SUBAPPLICATION Uebung_011f_ROUND_AR_AX (* Wie Uebung_011f_AX, aber mit OSCAT ROUND_AR dazwischen (rundet auf N Nachkommastellen) *)
  (* Standard: 61499-2; Description: Copyright (c) 2026 Meisterschulen am Ostbahnhof This program and the accompanying materials are made available under the terms of the Eclipse Public License 2.0 which is available at https://www.eclipse.org/legal/epl-2.0/ SPDX-License-Identifier: EPL-2.0 *)
  (* Version 1.0, 2026-10-09, Franz Höpfinger, Meisterschulen am Ostbahnhof, initial API and implementation and/or initial documentation *)
  PACKAGE Uebungen;
  IMPORT Uebungen::const::UT::DefaultPool_Numeric::InputNumber_I3_N;
  IMPORT Uebungen::const::UT::DefaultPool_Numeric::OutputNumber_N3_N;
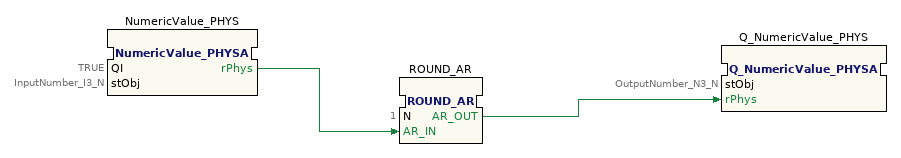
  (* Beispiel: I3-Eingabe -500.00 -> rPhys=-500.0 -> ROUND_AR (N=1) -> -500.0 -> Q_NumericValue_PHYS(N3) -> N3 zeigt -500.00. *)
  FBS
    NumericValue_PHYS : isobus::UT::io::NumericValue::NumericValue_PHYSA(QI := TRUE, stObj := InputNumber_I3_N);
    ROUND_AR : OSCAT_adapter::Mathematical::ROUND_AR(N := 1); (* Rundet auf N Nachkommastellen *)
    Q_NumericValue_PHYS : isobus::UT::Q::Q_NumericValue_PHYSA(stObj := OutputNumber_N3_N);
  END_FBS
  ADAPTER_CONNECTIONS
    NumericValue_PHYS.rPhys TO ROUND_AR.AR_IN;
    ROUND_AR.AR_OUT TO Q_NumericValue_PHYS.rPhys;
  END_CONNECTIONS
END_SUBAPPLICATION
